// TIA Portal V18 export
FUNCTION "AHUIAQDemand" : Void   // FC60009, LAD
{ S7_Optimized_Access := 'TRUE' }
VERSION : 0.1
// stored: AutoNumber false, IsIECCheckEnabled false, SetENOAutomatically false, UDAEnableTagReadback false
   VAR_INPUT
      iUnitID : Int;
      cRegState : Byte;
      rActual : Real;
      rSetPoint : Real;
   END_VAR
   VAR_OUTPUT
      rDemand : Real;
   END_VAR
BEGIN
END_FUNCTION
